{attribute 'qualified_only'}
{attribute 'strict'}
TYPE HomingMode :
(
	eManual := 1,
	eAuto := 2
);
END_TYPE

(* stored: Version 1.1.0.1, ProductVersion 3.1.4024.6
   DUT HomingMode: Id {d8bf8b35-991e-451c-bbae-ad3e4db53452} *)
